Universal Robots PolyScope program: close_gripper.urp

Program close_gripper (installation=default directory=/programs/usbdisk createdIn=5.11.0.108249 lastSavedIn=5.11.0.108249 robotSerialNumber=20215300716)
Calibrated DH parameters: a=[-0.000028, -0.208258, -0.213299, -0.000059, -0.000159, 0]; d=[0.151933, 47.085825, -45.764842, -1.189709, 0.085442, 0.092078]; alpha=[1.570477, 0.00269, 0.003865, 1.571648, -1.571757, 0]; deltaTheta=[0, 0.546481, -0.522554, -0.023924, 0.000003, 0]
Robot Program (runOnlyOnce=false)
  URCap Zimmer (Z_Gripper_C, Zimmer Group) dataModel(gripper_installation_scheme=257, gripper_number=3, program_number=2, program_name=Z_Grip, program_settings=264)
